// TwinCAT 3 PLC project SPS
// ProgramVersion: 3.1.4024.0
// libraries:
//   Tc2_Standard, * (Beckhoff Automation GmbH)
//   Tc2_System, * (Beckhoff Automation GmbH)
//   Tc3_Module, * (Beckhoff Automation GmbH)
// project tree:
//   DUTs/ E_STATE_AMPEL.TcDUT, E_State_Linie.TcDUT, E_State_Rob.TcDUT, E_State_Transport.TcDUT
//   GVLs/ GVL.TcGVL
//   / PlcTask.TcTTO
//   POUs/ MAIN.TcPOU
//   POUs/Rob_Steuerung/ Hauptablauf.TcPOU, Kommunikation.TcPOU
//   POUs/Transport/ Ampel.TcPOU, Linie.TcPOU, Transport.TcPOU
// real-time tasks:
//   TASK PlcTask: cycle T#10ms, priority 20, ADS port 350
//   TASK PlcTask1: cycle T#10ms, priority 21, ADS port 351

CONFIGURATION SPS
    RESOURCE PLC ON TwinCAT3
        TASK PlcTask(INTERVAL := T#10ms, PRIORITY := 21);
        PROGRAM MAIN WITH PlcTask : MAIN;
    END_RESOURCE
END_CONFIGURATION

// ---- DUTs/E_STATE_AMPEL.TcDUT
{attribute 'qualified_only'}
{attribute 'strict'}
TYPE E_STATE_AMPEL :
(
	OFF,
	RED,
	GREEN,
	YELLOW,
	BLINK,
	ALL
);
END_TYPE

// ---- DUTs/E_State_Linie.TcDUT
{attribute 'qualified_only'}
{attribute 'strict'}
TYPE E_State_Linie :
(
	IDLE,
	INIT,
	START,
	OPEN_MIDLE,
	CLOSE_MIDLE,
	OPEN_START,
	CLOSE_START,
	WAIT_MIDLE,
	WAIT_START,
	DONE
	
);
END_TYPE

// ---- DUTs/E_State_Rob.TcDUT
{attribute 'qualified_only'}
{attribute 'strict'}
TYPE E_State_Rob :
(
	IDLE,
	INIT,
	WAIT_CRATE,
	START_BIN_PICKING,
	START_QUALITY,
	GET_NEW_CRATE,
	MOVE_TO_QUALI,
	QUALI_PICTURE,
	WAIT_CRATE_2,
	PLACE_GOOD,
	PLACE_BAD,
	DONE
);
END_TYPE

// ---- DUTs/E_State_Transport.TcDUT
{attribute 'qualified_only'}
{attribute 'strict'}
TYPE E_State_Transport :
(
    IDLE,
    INIT,
    WORK

);
END_TYPE

// ---- GVLs/GVL.TcGVL
{attribute 'qualified_only'}
VAR_GLOBAL
	
	//Taster
	bStart: BOOL;
	bQuitieren: BOOL;
	bStop: BOOL;
	
	//Sensoren
	//Sotieranlage hat zwei linien 1 Zuliferung der Teile 2 Abtransport
	bB1_1 : BOOL; //Sensor Vorne
	bB1_2 :BOOL;  //Sensor Mitte
	bB1_3:BOOL; //Sensor Ende
	
	bB2_1 : BOOL; //Sensor Vorne
	bB2_2 :BOOL;  //Sensor Mitte
	bB2_3:BOOL; //Sensor Ende
	
	//Aktoren
	//Sotieranlage hat zwei linien 1 Zuliferung der Teile 2 Abtransport
	bM1_1 :BOOL; //Rollenstopper Vorne
	bM1_2 :BOOL; //Rollenstopper Mitte
	
	
	bM2_1 :BOOL; //Rollenstopper Vorne
	bM2_2 :BOOL; //Rollenstopper Mitte
	
	
	//Ampeln
	//Sotieranlage hat zwei linien 1 Zuliferung der Teile 2 Abtransport
	bP1_1R:BOOL; //Ampel Rot
	bP1_1Y:BOOL; //Ampel Gelb
	bP1_1G:BOOL; //Ampel Gruen
	
	bP1_3R:BOOL; //Ampel Rot
	bP1_3Y:BOOL; //Ampel Gelb
	bP1_3G:BOOL; //Ampel Gruen
	
	bP2_1R:BOOL; //Ampel Rot
	bP2_1Y:BOOL; //Ampel Gelb
	bP2_1G:BOOL; //Ampel Gruen
	
	bP2_3R:BOOL; //Ampel Rot
	bP2_3Y:BOOL; //Ampel Gelb
	bP2_3G:BOOL; //Ampel Gruen	
	
	//Einstellungswerte
	iKisten_Kap:INT :=6; //Kapazität der Ablage
	
	// SPS → Roboter
	bRobot_Start 			   :BOOL;    //Startet Roboter
	bRobot_Start_BinPicking    : BOOL;  // Starte Bildaufnahme + Greifen
	bRobot_Start_QualityCheck  : BOOL;  // Bewege Teil zur Quali-Kamera
	bRobot_Place_Good_Part     : BOOL;  // Lege Gutteil in Kiste Strecke 2
	bRobot_Dispose_Bad_Part    : BOOL;  // Entsorge Schlechtteil
	
	// Roboter → SPS  
	bRobot_Ready              : BOOL;  // Bereit für neuen Auftrag
	bRobot_BinPicking_Done    : BOOL;  // Greifen abgeschlossen
	bRobot_At_Quality_Pos     : BOOL;  // Teil bei Quali-Kamera positioniert
	bRobot_Part_Placed        : BOOL;  // Teil abgelegt/entsorgt
	bRobot_Box_Empty          : BOOL;  // Kiste ist leer (von Kamera erkannt)
	bRobot_Error              : BOOL;  // Fehler aufgetreten
	wRobot_Error_Code         : WORD;  // Fehlercode ?
	
	
	// SPS → Kamera
	bQuality_Take_Picture     : BOOL;  // Mache Foto
	
	// Kamera → SPS
	bQuality_Ready            : BOOL;  // Bereit für Foto
	bQuality_Picture_Done     : BOOL;  // Foto aufgenommen
	bQuality_Result_Good      : BOOL;  // Teil ist OK
	bQuality_Error            : BOOL;  // Kamera-Fehler
	wQuality_Error_Code       : WORD;  // Fehlercode ?
END_VAR

// ---- POUs/MAIN.TcPOU
PROGRAM MAIN
VAR
	Transport: Transport;
	RS_Start_Stop  : RS;
	bKiste_Leer:BOOL:=FALSE;
	estate_Transport:E_State_Transport;
	ipart_counter:INT:=0;
	estate_Ampel_1_1 : E_STATE_AMPEL;
	estate_Ampel_1_2 : E_STATE_AMPEL;
	estate_Ampel_2_1 : E_STATE_AMPEL;
	estate_Ampel_2_2 : E_STATE_AMPEL;
	Ampel_1_1: Ampel;
	Ampel_1_2: Ampel;
	Ampel_2_1: Ampel;
	Ampel_2_2: Ampel;
	Bin_Picking: Hauptablauf;
END_VAR


RS_Start_Stop(SET:=GVL.bStart,RESET1:=GVL.bStop);

Transport( 
	bStart:= RS_Start_Stop.Q1, 
	bStop:= NOT(RS_Start_Stop.Q1),
	bSensor_Vorne_1:= GVL.bB1_1, 
	bSensor_Mitte_1:= GVL.bB1_2, 
	bSensor_Hinten_1:= GVL.bB1_3, 
	bSensor_Vorne_2:= GVL.bB2_1, 
	bSensor_Mitte_2:= GVL.bB2_2, 
	bSensor_Hinten_2:= GVL.bB2_3,  
	bKisteLeer:= bKiste_Leer, 
	estate=> estate_Transport, 
	estate_Ampel_1_1=> estate_Ampel_1_1,
	estate_Ampel_1_2=> estate_Ampel_1_2,
	estate_Ampel_2_1=> estate_Ampel_2_1,
	estate_Ampel_2_2=> estate_Ampel_2_2,    
	Rollenstopper_L1_1=> GVL.bM1_1, 
	Rollenstopper_L1_2=> GVL.bM1_2, 
	Rollenstopper_L2_1=> GVL.bM2_1, 
	Rollenstopper_L2_2=> GVL.bM2_2, 
	ipart_counter:= ipart_counter);
	
Bin_Picking(bStart:=RS_Start_Stop.Q1,bStop:=NOT(RS_Start_Stop.Q1), bchest_empty:=bKiste_Leer,Kiste_Zuliefern:=GVL.bB1_2,Kiste_Abtransport:=GVL.bB2_2,part_counter:=ipart_counter);
	
	

Ampel_1_1(e_state_ample:=estate_Ampel_1_1 , red=>GVL.bP1_1R , yellow=>GVL.bP1_1Y , green=>GVL.bP1_1G );
Ampel_1_2(e_state_ample:=estate_Ampel_1_2 , red=>GVL.bP1_3R , yellow=>GVL.bP1_3Y , green=>GVL.bP1_3G );
Ampel_2_1(e_state_ample:=estate_Ampel_2_1 , red=>GVL.bP2_1R , yellow=>GVL.bP2_1Y , green=>GVL.bP2_1G );
Ampel_2_2(e_state_ample:=estate_Ampel_2_2 , red=>GVL.bP2_3R , yellow=>GVL.bP2_3Y , green=>GVL.bP2_3G );

END_PROGRAM

// ---- POUs/Transport/Transport.TcPOU
FUNCTION_BLOCK Transport
VAR_INPUT
	bStart:BOOL;
	bStop:BOOL;
	bSensor_Vorne_1 :BOOL;
	bSensor_Mitte_1 :BOOL;
	bSensor_Hinten_1 :BOOL;
	bSensor_Vorne_2 :BOOL;
	bSensor_Mitte_2 :BOOL;
	bSensor_Hinten_2 :BOOL;
	
	
	
END_VAR
VAR_OUTPUT
	estate: E_State_Transport;
	estate_Ampel_1_1 : E_STATE_AMPEL;
	estate_Ampel_1_2 : E_STATE_AMPEL;
	estate_Ampel_2_1 : E_STATE_AMPEL;
	estate_Ampel_2_2 : E_STATE_AMPEL;
	Rollenstopper_L1_1:BOOL;
	Rollenstopper_L1_2:BOOL;
	Rollenstopper_L2_1:BOOL;
	Rollenstopper_L2_2:BOOL;
	
END_VAR
VAR_IN_OUT
	ipart_counter :INT;
	bKisteLeer:BOOL;
END_VAR

VAR
	FB_L1:Linie;
	FB_L2:linie;
END_VAR

FB_L1(bSensor_Vorne:=bSensor_Vorne_1,
	bSensor_Mitte:=bSensor_Mitte_1,
	bSensor_Hinten:=bSensor_Hinten_1,
	bRollenStopper_Vorne=>Rollenstopper_L1_1,
	bRollenStopper_Mitte=>Rollenstopper_L1_2,
	estate_A1=>estate_Ampel_1_1,
	estate_A2=>estate_Ampel_1_2);
	
FB_L2(bSensor_Vorne:=bSensor_Vorne_2,
	bSensor_Mitte:=bSensor_Mitte_2,
	bSensor_Hinten:=bSensor_Hinten_2,
	bRollenStopper_Vorne=>Rollenstopper_L2_1,
	bRollenStopper_Mitte=>Rollenstopper_L2_2,
	estate_A1=>estate_Ampel_2_1,
	estate_A2=>estate_Ampel_2_2);



CASE eState OF

    E_State_Transport.IDLE:
        IF bStart AND NOT bStop THEN
            eState := E_State_Transport.INIT;
        END_IF

    E_State_Transport.INIT:
		FB_L1.bEnable:=TRUE;
		FB_L2.bEnable:=TRUE;
        IF bStart THEN
            eState := E_State_Transport.WORK;
        END_IF

    E_State_Transport.WORK:
	
        IF bKisteLeer THEN
			FB_L1.bStart:=TRUE;
			IF FB_L1.estate = E_State_Linie.DONE THEN
				bKisteLeer:=FALSE;
				FB_L1.bStart:=FALSE;
			END_IF
		END_IF
		
        IF ipart_counter >= GVL.iKisten_Kap THEN
			FB_L2.bStart:=TRUE;
			IF FB_L2.estate = E_State_Linie.DONE THEN
				ipart_counter := 0;
				FB_L2.bStart:=FALSE;
			END_IF
        END_IF

END_CASE

IF bStop THEN
	FB_L1.bStart:=FALSE;
	FB_L2.bStart:=FALSE;
	FB_L1.bEnable:=FALSE;
	FB_L2.bEnable:=FALSE;
	estate:= E_State_Transport.IDLE;
END_IF

END_FUNCTION_BLOCK

// ---- POUs/Transport/Linie.TcPOU
FUNCTION_BLOCK Linie
VAR_INPUT
	bEnable:BOOL;
	bStart:BOOL;
	bSensor_Vorne :BOOL;
	bSensor_Mitte :BOOL;
	bSensor_Hinten :BOOL;
END_VAR
VAR_OUTPUT
	bRollenStopper_Vorne :BOOL;
	bRollenStopper_Mitte :BOOL;	
	estate : E_State_Linie;
	estate_A1 :E_STATE_AMPEL;
	estate_A2 :E_STATE_AMPEL;
END_VAR
VAR
	T_enable:BOOL;
    tTimer : TON; // Timer Variable
END_VAR


tTimer(IN:=T_enable, PT:=T#1S);

IF NOT bEnable THEN
    eState := E_State_Linie.IDLE;
END_IF

CASE eState OF
    E_State_Linie.IDLE:
	
        IF bEnable THEN
            eState := E_State_Linie.INIT;
        END_IF

    E_State_Linie.INIT:

		//Ampel 1 Umschalten
		IF NOT bSensor_Vorne THEN
			estate_A1 :=E_STATE_AMPEL.YELLOW;
		ELSE
			estate_A1 :=E_STATE_AMPEL.GREEN;
		END_IF
		//Ampel 2 Umschalten
		IF  bSensor_Hinten THEN
			estate_A2 :=E_STATE_AMPEL.YELLOW;
		ELSE
			estate_A2 :=E_STATE_AMPEL.GREEN;
		END_IF
		
		IF NOT bSensor_Mitte AND bSensor_Vorne THEN
			eState := E_State_Linie.OPEN_START;
		ELSIF NOT bSensor_Mitte AND NOT bSensor_Vorne THEN
		 	eState:=E_State_Linie.WAIT_START;
		END_IF
		
	    IF bStart THEN
			eState:=E_State_Linie.START;
		END_IF
		
	E_State_Linie.START:
		//Ampel 1 Umschalten
		IF NOT bSensor_Vorne THEN
			estate_A1 :=E_STATE_AMPEL.YELLOW;
		ELSE
			estate_A1 :=E_STATE_AMPEL.GREEN;
		END_IF
		//Ampel 2 Umschalten
		
		IF  bSensor_Hinten THEN
			estate_A2 :=E_STATE_AMPEL.YELLOW;
		ELSE
			estate_A2 :=E_STATE_AMPEL.GREEN;
		END_IF
	
		IF bSensor_Hinten AND bSensor_Mitte THEN
			eState := E_State_Linie.WAIT_MIDLE;		
		ELSIF NOT bSensor_Hinten AND bSensor_Mitte THEN
			eState := E_State_Linie.OPEN_MIDLE;
		END_IF
		
	E_State_Linie.WAIT_MIDLE:
	
		estate_A2 :=E_STATE_AMPEL.RED;
		IF NOT bSensor_Hinten THEN
			eState := E_State_Linie.OPEN_MIDLE;
		END_IF

    E_State_Linie.OPEN_MIDLE:
	
		bRollenStopper_Mitte:=TRUE;
		IF NOT bSensor_Mitte THEN
			T_enable:=TRUE;
		END_IF
        IF tTimer.Q THEN
            eState := E_State_Linie.CLOSE_MIDLE;
			T_enable:=FALSE;
        END_IF

    E_State_Linie.CLOSE_MIDLE:
	
		bRollenStopper_Mitte:=FALSE;
        IF NOT bSensor_Mitte AND bSensor_Vorne THEN
            eState := E_State_Linie.OPEN_START;
		ELSIF NOT bSensor_Mitte AND NOT bSensor_Vorne THEN
			eState := E_State_Linie.WAIT_START;
        END_IF
		
	E_State_Linie.WAIT_START:
	
		estate_A1 :=E_STATE_AMPEL.RED;
        IF bSensor_Vorne THEN
            eState := E_State_Linie.OPEN_START;
        END_IF
		
    E_State_Linie.OPEN_START:
		bRollenStopper_Vorne:=TRUE;
		IF NOT bSensor_Vorne THEN
			T_enable:=TRUE;
		END_IF
        IF tTimer.Q THEN
            eState := E_State_Linie.CLOSE_START;
			T_enable:=FALSE;
        END_IF
		
    E_State_Linie.CLOSE_START:
	
		bRollenStopper_Vorne:=FALSE;
		IF bSensor_Mitte THEN
        	eState := E_State_Linie.DONE;
		END_IF	

    E_State_Linie.DONE:
    eState := E_State_Linie.IDLE;
	
END_CASE

END_FUNCTION_BLOCK

// ---- POUs/Transport/Ampel.TcPOU
FUNCTION_BLOCK Ampel
VAR_INPUT
	e_state_ample : E_STATE_AMPEL;
END_VAR
VAR_OUTPUT
	red:BOOL;
	yellow:BOOL;
	green:BOOL;
END_VAR
VAR
END_VAR

CASE e_state_ample OF
	
	E_STATE_AMPEL.OFF:
		red:=FALSE;
		green:=FALSE;
		yellow:=FALSE;
		
	E_STATE_AMPEL.ALL:
		red:=TRUE;
		green:=TRUE;
		yellow:=TRUE;
	
	E_STATE_AMPEL.RED:
		red:=TRUE;
		green:=FALSE;
		yellow:=FALSE;
		
	E_STATE_AMPEL.YELLOW:
		red:=FALSE;
		green:=FALSE;
		yellow:=TRUE;
		
	E_STATE_AMPEL.GREEN:
		red:=FALSE;
		green:=TRUE;
		yellow:=FALSE;
			
		
END_CASE

END_FUNCTION_BLOCK

// ---- POUs/Rob_Steuerung/Hauptablauf.TcPOU
FUNCTION_BLOCK Hauptablauf
VAR_INPUT
	bStart: BOOL;
	bStop: BOOL; 
	Kiste_Zuliefern:BOOL;
	Kiste_Abtransport:BOOL;
END_VAR
VAR_OUTPUT
END_VAR
VAR
	eState_Robot: E_STATE_ROB;
	fbBoxEmptyPos : R_TRIG;
END_VAR

VAR_IN_OUT
	part_counter :INT;
	bchest_empty :BOOL;
END_VAR

// Flankenerkennung
fbBoxEmptyPos(CLK := GVL.bRobot_Box_Empty);

IF fbBoxEmptyPos.Q THEN
	bchest_empty:=TRUE;
END_IF

//Schrittkette
CASE eState_Robot OF
	
	E_State_Rob.IDLE:
		// Initialisierung
		GVL.bRobot_Start_BinPicking := FALSE;
		GVL.bRobot_Start_QualityCheck := FALSE;
		GVL.bRobot_Place_Good_Part := FALSE;
		GVL.bRobot_Dispose_Bad_Part := FALSE;
		GVL.bQuality_Take_Picture := FALSE;
		
		// Warten bis System bereit
		IF bStart THEN
			eState_Robot := E_State_Rob.INIT;
		END_IF
		
	E_State_Rob.INIT: 
	GVL.bRobot_Start:= TRUE;		
	IF GVL.bRobot_Ready THEN
			eState_Robot := E_State_Rob.WAIT_CRATE;
	END_IF
	
	E_State_Rob.WAIT_CRATE:
		IF Kiste_Zuliefern THEN  
			eState_Robot := E_State_Rob.START_BIN_PICKING;
		END_IF
	
	E_State_Rob.START_BIN_PICKING:
		// Bin-Picking starten
		GVL.bRobot_Start_BinPicking := TRUE;
		
		// Warten auf Roboter-Rückmeldung
		IF GVL.bRobot_BinPicking_Done THEN
			GVL.bRobot_Start_BinPicking := FALSE;
			
			IF bchest_empty THEN				
				eState_Robot := E_State_Rob.GET_NEW_CRATE;
			ELSE
				eState_Robot := E_State_Rob.MOVE_TO_QUALI;
			END_IF
		ELSIF GVL.bRobot_Error THEN
			// Fehlerbehandlung
			GVL.bRobot_Start_BinPicking := FALSE;
			eState_Robot := E_State_Rob.INIT;  // Oder zu Fehler-State
		END_IF
	
	E_State_Rob.MOVE_TO_QUALI:
		// Roboter zur Qualitätsprüfung bewegen
		GVL.bRobot_Start_QualityCheck := TRUE;
		
		IF GVL.bRobot_At_Quality_Pos THEN
			GVL.bRobot_Start_QualityCheck := FALSE;
			eState_Robot := E_State_Rob.START_QUALITY;
		END_IF
	
	E_State_Rob.GET_NEW_CRATE:
		IF Kiste_Zuliefern AND NOT bchest_empty THEN
			eState_Robot := E_State_Rob.START_BIN_PICKING;
		END_IF
	
	E_State_Rob.START_QUALITY:
		// Roboter ist an Qualitätsposition, Foto machen
		GVL.bQuality_Take_Picture := TRUE;
		
		IF GVL.bQuality_Picture_Done THEN
			GVL.bQuality_Take_Picture := FALSE;
			eState_Robot := E_State_Rob.QUALI_PICTURE;
		ELSIF GVL.bQuality_Error THEN
			// Qualitätsfehler
			GVL.bQuality_Take_Picture := FALSE;
			eState_Robot := E_State_Rob.INIT;
		END_IF
	
	E_State_Rob.QUALI_PICTURE:
		// Qualitätsergebnis auswerten
		IF GVL.bQuality_Result_Good AND Kiste_Abtransport THEN
			eState_Robot := E_State_Rob.PLACE_GOOD;
		ELSIF GVL.bQuality_Result_Good AND NOT Kiste_Abtransport THEN
			eState_Robot := E_State_Rob.WAIT_CRATE_2;
		ELSE
			eState_Robot := E_State_Rob.PLACE_BAD;
		END_IF
		
	E_State_Rob.WAIT_CRATE_2:
		IF Kiste_Abtransport THEN
			eState_Robot := E_State_Rob.PLACE_GOOD;
		END_IF
	
	E_State_Rob.PLACE_GOOD:
		// Gutteil in Abtransportkiste legen
		GVL.bRobot_Place_Good_Part := TRUE;
		IF GVL.bRobot_Part_Placed THEN
			GVL.bRobot_Place_Good_Part := FALSE;
			eState_Robot := E_State_Rob.DONE;
			part_counter := part_counter +1;
		ELSIF GVL.bRobot_Error THEN
			// Ablegefehler
			GVL.bRobot_Place_Good_Part := FALSE;
			eState_Robot := E_State_Rob.INIT;
		END_IF
	
	E_State_Rob.PLACE_BAD:
		// Schlechtteil entsorgen
		GVL.bRobot_Dispose_Bad_Part := TRUE;
		
		IF GVL.bRobot_Part_Placed THEN
			GVL.bRobot_Dispose_Bad_Part := FALSE;
			eState_Robot := E_State_Rob.DONE;
		ELSIF GVL.bRobot_Error THEN
			// Entsorgungsfehler
			GVL.bRobot_Dispose_Bad_Part := FALSE;
			eState_Robot := E_State_Rob.INIT;
		END_IF
	
	E_State_Rob.DONE:
		// Zyklus abgeschlossen, prüfen ob weitere Teile
		IF GVL.bRobot_Ready THEN
			IF Kiste_Zuliefern THEN  // Noch Kiste da
				eState_Robot := E_State_Rob.START_BIN_PICKING;
			ELSE
				eState_Robot := E_State_Rob.WAIT_CRATE;
			END_IF
		END_IF

ELSE
	// Unbekannter Zustand - Reset
	eState_Robot := E_State_Rob.INIT;
	
END_CASE

// Stop-Button Behandlung
IF bStop THEN
	eState_Robot := E_State_Rob.INIT;
	// Alle Ausgänge zurücksetzen
	GVL.bRobot_Start:= FALSE;
	GVL.bRobot_Start_BinPicking := FALSE;
	GVL.bRobot_Start_QualityCheck := FALSE;
	GVL.bRobot_Place_Good_Part := FALSE;
	GVL.bRobot_Dispose_Bad_Part := FALSE;
	GVL.bQuality_Take_Picture := FALSE;
END_IF

END_FUNCTION_BLOCK

// ---- POUs/Rob_Steuerung/Kommunikation.TcPOU
FUNCTION_BLOCK Kommunikation
VAR_INPUT
END_VAR
VAR_OUTPUT
END_VAR
VAR
END_VAR

END_FUNCTION_BLOCK
